// TwinCAT 3 PLC project CNCControl
// ProgramVersion: 3.1.4022.4
// libraries:
//   Tc2_EthernetIP, * (Beckhoff Automation GmbH)
//   Tc2_IoFunctions, * (Beckhoff Automation GmbH)
//   Tc2_Math, * (Beckhoff Automation GmbH)
//   Tc2_Standard, * (Beckhoff Automation GmbH)
//   Tc2_System, * (Beckhoff Automation GmbH)
//   Tc2_Utilities, * (Beckhoff Automation GmbH)
//   Tc3_Module, * (Beckhoff Automation GmbH)
// project tree:
//   DUTs/ E_CIA402State.TcDUT, E_PIDOptimizationStage.TcDUT, E_PIDOptimizationType.TcDUT
//   / EveryHundredMilliseconds.TcTTO, EveryMS.TcTTO (not stored), MainCNCControl.TcTTO (not stored)
//   GVLs/ Constants.TcGVL
//   POUs/ MAIN.TcPOU
//   POUs/SpindleSpeed/ AnalogDemandedSpeedCalculator.TcPOU (not stored), AnalogPrescaledSpeedCalculator.TcPOU, DemandedSpeedInterface.TcIO (not stored), DemandedSpeedTask.TcPOU, PWMDemandedSpeedCalculator.TcPOU, SpindleSpeedCalculator.TcPOU (not stored)
//   POUs/Spindle/ SpindleCIA402Velocity.TcPOU, SpindleController.TcIO, SpindleDeltaVFDOverEIP.TcPOU, SpindleKEBWithEncoder.TcPOU
//   POUs/Utilities/ FB_FreqMeasure.TcPOU, FB_MovingAverageUInt.TcPOU (not stored), FB_MovingAverageReal.TcPOU, FB_OptimizePID.TcPOU (not stored), FB_ScaleBetween.TcPOU (not stored)
//   POUs/Vacuum/ VacuumATV71Ethercat.TcPOU, FB_GetVacuumAMSID.TcPOU, ToshibaP9VacuumPressureGetter.TcPOU, VacuumController.TcIO (not stored)
// real-time tasks:
//   TASK EveryHundredMilliseconds: cycle T#100000us, priority 10, ADS port 350
//   TASK MainCNCControl: cycle T#1ms, priority 6, ADS port 351
//   TASK EveryMS: cycle T#1ms, priority 4, ADS port 352
// I/O:
//   DEVICE Device 1 (EtherCAT), AmsNetId 192.168.1.51.2.1
//     Box 16 (ATV71 EtherCAT) [ATV71 EtherCAT]
//     HITECO UE-1F 6.6 Spindle [KEB_F6_drive_unit_EtherCAT (MDP)]
//       modules: Module 1 (Spindle_Profile)
//     Term 1 (EK1100) [EK1100 EtherCAT Coupler (2A E-Bus)]
//       Term 9 (EL2809) [EL2809 16Ch. Dig. Output 24V, 0.5A]
//       Term 3 (EL1502) [EL1502 2Ch. +/- Counter 24V, 100kHz]
//       Term 4 (EL1809) [EL1809 16Ch. Dig. Input 24V, 3ms]
//       Term 26 (EL6070) [EL6070 1Ch. Licensing-Terminal]
//       Term 17 (EL9110) [EL9110 Power Supplier with LED (24V, Diagnostics)]
//       Term 19 (EL3161) [EL3161 1Ch. Ana. Input 0-10V]
//       Term 12 (EL9011) [EL9011 End Terminal]
//   DEVICE Device 2 (TC3 EIP Scanner), AmsNetId 192.168.1.51.3.1
//     Box 12 (Nitra CMV EtherNet/IP) // <INFO> </INFO> <EDS> C:\TwinCAT\3.1\Config\Io\EtherNetIP\nitraethernetip.eds </EDS>
//     Box 13 (IPE001Z) (disabled) // <INFO> </INFO> <EDS> C:\TwinCAT\3.1\Config\Io\EtherNetIP\IPE001Z_AS1.eds </EDS>
//     Box 2 (CMM-EIP01) (disabled) // <INFO> </INFO> <EDS> C:\TwinCAT\3.1\Config\Io\EtherNetIP\031F000C010400010001.eds </EDS>
// variable links:
//   CNCControl/CNCControl Instance <-> Device 1 (EtherCAT)/Box 16 (ATV71 EtherCAT)
//     MainCNCControl Inputs/MAIN.VacuumControl.iAnalogInput2ScaledValue <-> Inputs/MAIN.VacuumControl.iAnalogInput2ScaledValue
//     MainCNCControl Inputs/MAIN.VacuumControl.iOutputFrequency <-> Inputs/MAIN.VacuumControl.iOutputFrequency
//     MainCNCControl Inputs/MAIN.VacuumControl.iOutputVelocity <-> Inputs/MAIN.VacuumControl.iOutputVelocity
//     MainCNCControl Inputs/MAIN.VacuumControl.iPIDRegulatorFeedback <-> Inputs/MAIN.VacuumControl.iPIDRegulatorFeedback
//     MainCNCControl Inputs/MAIN.VacuumControl.iPIDRegulatorOutput <-> Inputs/MAIN.VacuumControl.iPIDRegulatorOutput
//     MainCNCControl Inputs/MAIN.VacuumControl.iStatusWord <-> Inputs/MAIN.VacuumControl.iStatusWord
//     MainCNCControl Outputs/MAIN.VacuumControl.oMotorFrequency <-> Outputs/MAIN.VacuumControl.oMotorFrequency
//     MainCNCControl Outputs/MAIN.VacuumControl.oVacuumControl <-> Outputs/MAIN.VacuumControl.oVacuumControl
//     MainCNCControl Outputs/MAIN.VacuumControl.oVacuumPressureRequested <-> Outputs/MAIN.VacuumControl.oVacuumPressureRequested
//   CNCControl/CNCControl Instance <-> Device 1 (EtherCAT)/HITECO UE-1F 6.6 Spindle
//     MainCNCControl Inputs/MAIN.SpindleControl.iActualVelocity <-> Module 1 (Spindle_Profile)/Inputs/velocity actual value [0x606C.0]
//     MainCNCControl Inputs/MAIN.SpindleControl.iEncoderErrorState <-> Module 1 (Spindle_Profile)/Inputs/ec01: error encoder interface [0x2801.0]
//     MainCNCControl Inputs/MAIN.SpindleControl.iStatusWord <-> Module 1 (Spindle_Profile)/Inputs/statusword [0x6041.0]
//     MainCNCControl Outputs/MAIN.SpindleControl.oControlWord <-> Module 1 (Spindle_Profile)/Outputs/controlword [0x6040.0]
//     MainCNCControl Outputs/MAIN.SpindleControl.oDigitalInputs <-> Module 1 (Spindle_Profile)/Outputs/di02: dig. input ext. src. [0x3202.0]
//     MainCNCControl Outputs/MAIN.SpindleControl.oTargetVelocity <-> Module 1 (Spindle_Profile)/Outputs/vl target velocity [0x6042.0]
//   CNCControl/CNCControl Instance <-> Device 1 (EtherCAT)/Term 1 (EK1100)/Term 3 (EL1502)
//     EveryHundredMilliseconds Inputs/SpindleSpeedCalculator.CounterValue <-> CNT Inputs Channel 1/Counter value
//   CNCControl/CNCControl Instance <-> Device 1 (EtherCAT)/Term 1 (EK1100)/Term 4 (EL1809)
//     MainCNCControl Inputs/MAIN.iAirPressureSensor <-> Channel 1/MAIN.iPressureSensor
//     MainCNCControl Inputs/MAIN.iS1ToolPresence <-> Channel 5/MAIN.iS1ToolPresence
//     MainCNCControl Inputs/MAIN.iS2ColletOpen <-> Channel 4/MAIN.iS2ColletOpen
//     MainCNCControl Inputs/MAIN.iSpindleOverTemp <-> Channel 3/MAIN.iSpindleOverTemp
//     MainCNCControl Inputs/MAIN.iSpindleToolReleaseButton <-> Channel 2/MAIN.iSpindleToolReleaseButton
//   CNCControl/CNCControl Instance <-> Device 2 (TC3 EIP Scanner)/Box 12 (Nitra CMV EtherNet/IP)
//     MainCNCControl Outputs/MAIN.oValveControl <-> Connection 1 (Input/Output)/Outputs/MAIN.oValveControl

CONFIGURATION CNCControl
    RESOURCE PLC ON TwinCAT3
        TASK EveryHundredMilliseconds(INTERVAL := T#100000us, PRIORITY := 10);
        PROGRAM SpindleSpeedCalculator WITH EveryHundredMilliseconds : SpindleSpeedCalculator;
    END_RESOURCE
END_CONFIGURATION

// ---- DUTs/E_CIA402State.TcDUT
{attribute 'qualified_only'}
{attribute 'strict'}
TYPE E_CIA402State :
(
	Unknown_State,
	NotReadyToSwitchOn,
	SwitchOnDisabled,
	ReadyToSwitchOn,
	SwitchedOn,
	OperationEnabled,
	QuickStopActive,
	FaultReactionActive,
	Fault
);
END_TYPE

// ---- DUTs/E_PIDOptimizationStage.TcDUT
{attribute 'qualified_only'}
{attribute 'strict'}
TYPE E_PIDOptimizationStage :
(
	Init,
	RampingUp,
	RampingDown,
	Done
);
END_TYPE

// ---- DUTs/E_PIDOptimizationType.TcDUT
{attribute 'qualified_only'}
{attribute 'strict'}
TYPE E_PIDOptimizationType :
(
	NoOvershoot,
	SomeOvershoot,
	PessenIntegralRule
);
END_TYPE

// ---- GVLs/Constants.TcGVL
{attribute 'qualified_only'}
VAR_GLOBAL CONSTANT
	// One second in microseconds
	OneSecondInUs : UDINT := 1000000;
END_VAR

// ---- POUs/Spindle/SpindleController.TcIO
INTERFACE SpindleController

// Return the current speed of the spindle in RPM
METHOD GetSpeed : UDINT
VAR_INPUT
END_VAR
END_METHOD

// Start the Spindle running
METHOD Run : BOOL
END_METHOD

// Set the direction the spindle rotates in.
METHOD SetDirection : BOOL
VAR_INPUT
	// Set the spindle rotation direction
	Reverse : BOOL;
END_VAR
END_METHOD

// Set the target speed for the spindle.
METHOD SetSpeed : BOOL
VAR_INPUT
	Speed : UINT;
END_VAR
END_METHOD

// Stop the running spindle
METHOD Stop : BOOL
END_METHOD

END_INTERFACE

// ---- POUs/MAIN.TcPOU
PROGRAM MAIN
VAR
	{region "Air Pressure and Coolant"}
	// Air Pressure >90psi signal to PC pin 10
	oPCAirPressure AT %Q*: BOOL;
	// Air Pressure >90psi signal from sensor.  The sensor triggers as pressure is rising past 90psi
	iAirPressureSensor AT %I*: BOOL;
	// Control of NITRA Valves over ethernet/ip	 
	oValveControl AT %Q* : NitraValves; 
	// Turn on coolant signal from PC
	iPCCoolantOn AT %I* : BOOL;
	{endregion}
	{region "Vacuum"}
	VacuumControl: VacuumATV71Ethercat;
	 // Turn on vacuum signal from PC
	iPCVacuumOn AT %I* : BOOL;
	// Vacuum Pressure good output to PC Pin 7
	oPCVacuumPressureGood AT %Q*: BOOL;
	{endregion}
	{endregion}
	{endregion}
	{region "Spindle variables"}
	{region "Spindle Speed Handling"}
	// True if spindle is at less than 1 RPM
	SpindleStopped : BOOL;
	// Spindle stopped output to PC pin 1
	oPCSpindleStopped AT %Q* : BOOL;
	// Spindle within 5% of speed to PC Pin 28
	oPCSpindleSpeedOK AT %Q* : BOOL;
	{endregion}
	{region "Spindle Tool Change handling"}
	// Tool Release Button on Spindle
	iSpindleToolReleaseButton AT %I*: BOOL;
	// Tool Release from PC Pin 24
	iPCToolRelease AT %I*: BOOL;
	// Tool Presence to PC Pin 2
	oPCToolPresence AT %Q* : BOOL;
	// S1 Tool Presence sensor from the spindle
	iS1ToolPresence AT %I* : BOOL;
	// Collet Open to PC Pin 9
	oPCColletOpen AT %Q* : BOOL;
	// S2 Collet Open sensor from the spindle
	iS2ColletOpen AT %I* : BOOL;	 
	// Spindle over temperature to PC Pin 27
	oPCSpindleOverTemp AT %Q* : BOOL;
	// Spindle over temperature relay
	iSpindleOverTemp AT %I* : BOOL;
	// Turn spindle on input from PC
	iPCSpindleOn AT %I* : BOOL;
	SpindleControl : SpindleKEBWithEncoder;
	{endregion}
	{endregion}
	{region "Input Debouncers"}
	(* The 5V input has a ridiculously fast time - a few nanoseconds.
	   Therefore, we debounce it *)
	CoolantOnDebounced : TON;
	SpindleOnDebounced : TON;
	ToolReleaseDebounced : TON;	
	VacuumOnDebounced : TON;
	{endregion}
END_VAR
VAR CONSTANT
	// Minimum PSI at which vacuum holding is viable for workpiece
	GoodVacuumPressure : REAL := 10.0;
END_VAR

CoolantOnDebounced(IN := iPCCoolantOn, PT := T#3MS);
SpindleOnDebounced(IN := iPCSpindleOn, PT := T#3MS);
ToolReleaseDebounced(IN := iPCToolRelease, PT := T#3MS);
VacuumOnDebounced(IN := iPCVacuumOn, PT := T#3MS);

{region "Probe, Air Pressure, Coolant, Vacuum"}

// Pressure Control
	oPCAirPressure := iAirPressureSensor;

// Coolant control
	oValveControl.Coolant := CoolantOnDebounced.Q;

// Vacuum Control
	IF VacuumOnDebounced.Q THEN
		VacuumControl.Run();
	ELSE 
		VacuumControl.Stop();
	END_IF
	oPCVacuumPressureGood := VacuumControl.GetCurrentPressure() >= GoodVacuumPressure;

{endregion}
{region "Spindle handling"}
// Spindle Speed Handling
	// Spindle is stopped if it is under 1RPM
	SpindleStopped := SpindleSpeedCalculator.SpindleSpeed <= 1.0;
	oPCSpindleStopped := SpindleStopped;
	// Calculate whether spindle is up to speed.  We will only say it is up to speed if it is on.
	oPCSpindleSpeedOK := SpindleOnDebounced.Q AND_THEN (SpindleSpeedCalculator.SpindleSpeed  >= (0.95 * TO_REAL(DemandedSpeedTask.DemandedSpeed)));

// Spindle control handling
	 // NOTE: HSK-F63 spindles may not be spun while the tool is not present
	 IF NOT (SpindleOnDebounced.Q AND iS1ToolPresence) THEN
	 	SpindleControl.SetSpeed(0);
		SpindleControl.Stop();
	 ELSIF SpindleOnDebounced.Q AND iS1ToolPresence THEN	  
	 	SpindleControl.SetSpeed(DemandedSpeedTask.DemandedSpeed);
		SpindleControl.Run();
	 END_IF
		  
// Spindle Tool Change handling
	oPCToolPresence := iS1ToolPresence;
	oPCColletOpen := iS2ColletOpen;
	oPCSpindleOverTemp := iSpindleOverTemp;
	oValveControl.ToolRelease := (iAirPressureSensor AND_THEN SpindleStopped) AND_THEN (ToolReleaseDebounced.Q OR iSpindleToolReleaseButton); 		  

{endregion}		  
{endregion}

END_PROGRAM

// ---- POUs/Vacuum/VacuumATV71Ethercat.TcPOU
FUNCTION_BLOCK VacuumATV71Ethercat IMPLEMENTS  VacuumController
VAR_INPUT
END_VAR
VAR_OUTPUT
END_VAR
VAR
	// Vacuum Control Output
	oVacuumControl AT %Q* : ST_ATV71CommandWord;	
	// Vacuum Pressure requested from VFD - in tenths of a psi from 0 to 1450
	oVacuumPressureRequested AT %Q* : UINT;
		 
	{region "Input Vacuum Data"}
	iStatusWord AT %I* : UINT;
	{attribute 'BaseUnit' := '<RPM, 1, 0, 0>'}
	iOutputVelocity AT %I* : UINT;
	iAnalogInput2ScaledValue AT %I* : UINT;
	{attribute 'UserUnit' := '<Pressure, PSI, PSI, 6894.7572932, 0, centi>'}
	iPIDRegulatorFeedback AT %I* : UINT;
	iPIDRegulatorOutput AT %I* : UINT;
	{attribute 'BaseUnit' := '<Frequency, 0.1, 0, 0>'}
	iOutputFrequency AT %I* : UINT;
	{endregion}
	oMotorFrequency AT %Q* : UINT;
	//	PidOptimizer : FB_OptimizePID;
END_VAR

METHOD GetCurrentPressure : REAL
GetCurrentPressure := TO_REAL(iPIDRegulatorFeedback) / 100;
END_METHOD

METHOD Run : BOOL
oVacuumControl.Forward := TRUE;
oVacuumControl.Reverse := FALSE;
oVacuumControl.PidIntegralOff := FALSE;
	
	(* PID optimization
	IF VacuumOnDebounced.Q THEN
		IF NOT PidOptimizer.TuningDone THEN
			PidOptimizer(Enable := TRUE,
						 ProcessSetpoint := 2500,
						 ProcessValue := iAnalogInput2ScaledValue,
						 NumCycles := 10,
						 Reset := FALSE,
						 ControlLowVal := 5,
						 ControlHighVal := 60,
						 PIDType := E_PIDOptimizationType.FastRamp);
			oMotorFrequency := TO_UINT(PidOptimizer.ControlValue*10);
			IF PidOptimizer.TuningDone THEN
				ADSLOGLREAL(TC2_Utilities.ADSLOG_MSGTYPE_LOG, 'Kp value is %f', PidOptimizer.Kp);
				ADSLOGLREAL(TC2_Utilities.ADSLOG_MSGTYPE_LOG, 'Ki value is %f', PidOptimizer.Ki);
				ADSLOGLREAL(TC2_Utilities.ADSLOG_MSGTYPE_LOG, 'Kd value is %f', PidOptimizer.Kd);
				ADSLOGLREAL(TC2_Utilities.ADSLOG_MSGTYPE_LOG, 'Ku value is %f', PidOptimizer.Ku);
				ADSLOGLREAL(TC2_Utilities.ADSLOG_MSGTYPE_LOG, 'Tu value is %f', PidOptimizer.Tu);
			END_IF
		END_IF
	END_IF
	*)
END_METHOD

METHOD SetPressureRequired : BOOL
VAR_INPUT
	Pressure	: REAL;
END_VAR
oVacuumPressureRequested := TO_UINT(Pressure * 100);
END_METHOD

METHOD Stop : BOOL
oVacuumControl.Forward := FALSE;
oVacuumControl.Reverse := FALSE;
oVacuumControl.PidIntegralOff := FALSE;
END_METHOD

END_FUNCTION_BLOCK

// ---- POUs/Spindle/SpindleKEBWithEncoder.TcPOU
FUNCTION_BLOCK SpindleKEBWithEncoder EXTENDS SpindleCIA402Velocity IMPLEMENTS SpindleController
VAR_INPUT
END_VAR
VAR_OUTPUT
	// This represents the digital inputs of the KEB drive
	// Bit 0 resets the error state
	oDigitalInputs AT %Q* : UINT;
	// Encoder error state
	// Anything other than 0 is an error
	iEncoderErrorState AT %I* : UINT;
END_VAR
VAR
END_VAR

METHOD Stop : BOOL
// The 1024ppr encoder is only good to 12000rpm, so if you go faster, it will get an error that needs to be reset.
// This resets the error state (but only when the spindle is safely stopped)
IF iEncoderErrorState <> 0  AND GetState() = E_CIA402State.SwitchOnDisabled THEN
	oControlWord.FaultReset := TRUE;
ELSE
	oControlWord.FaultReset := FALSE;
	SUPER^.Stop();
END_IF
END_METHOD

END_FUNCTION_BLOCK

// ---- POUs/Spindle/SpindleCIA402Velocity.TcPOU
FUNCTION_BLOCK SpindleCIA402Velocity IMPLEMENTS SpindleController
VAR
	// CIA402 Control word
	oControlWord AT %Q*: ST_CIA402ControlWord;
	// CIA402 Status word
	iStatusWord AT %I*: UINT;
	// CIA402 actual velocity parameter
	iActualVelocity AT %I* : UDINT;
	// CIA402 target velocity
	oTargetVelocity AT %Q* : INT;
	// Forward/backward is specified by positive or negative speed
	VelocityMultiplier : INT := 1;
END_VAR

(* Return the current speed of the spindle in RPM*)
METHOD GetSpeed : UDINT
GetSpeed := iActualVelocity;
END_METHOD

METHOD GetState : E_CIA402State
VAR CONSTANT
	NotReadyToSwitchOnValue : UINT := 2#0000_0000_0000_0000;
	NotReadyToSwitchOnMask : UINT := 2#0000_0000_0100_1111;
	SwitchOnDisabledValue : UINT := 2#0000_0000_0100_0000;
	SwitchOnDisabledMask : UINT := NotReadyToSwitchOnMask;
	ReadyToSwitchOnValue : UINT := 2#0000_0000_0010_0001;
	ReadyToSwitchOnMask : UINT := 2#0000_0000_0110_1111;
	SwitchedOnValue : UINT := 2#0000_0000_0010_0011;
	SwitchedOnMask : UINT := ReadyToSwitchOnMask;
	OperationEnabledValue : UINT := 2#0000_0000_0010_0111;
	OperationEnabledMask : UINT := ReadyToSwitchOnMask;
	QuickStopActiveValue : UINT := 2#0000_0000_0000_0111;
	QuickStopActiveMask : UINT := ReadyToSwitchOnMask;
	FaultReactionActiveValue : UINT := 2#0000_0000_0000_1111;
	FaultReactionActiveMask : UINT := 2#0000_0000_0100_1111;
	FaultValue : UINT := 2#0000_0000_0000_1000;
	FaultMask : UINT := FaultReactionActiveMask;
END_VAR
IF (iStatusWord AND NotReadyToSwitchOnMask) = NotReadyToSwitchOnValue THEN
	GetState := E_CIA402State.NotReadyToSwitchOn;
ELSIF (iStatusWord AND SwitchOnDisabledMask) = SwitchOnDisabledValue THEN
	GetState := E_CIA402State.SwitchOnDisabled;
ELSIF (iStatusWord AND ReadyToSwitchOnMask) = ReadyToSwitchOnValue THEN
	GetState := E_CIA402State.ReadyToSwitchOn;
ELSIF (iStatusWord AND SwitchedOnMask) = SwitchedOnValue THEN
	GetState := E_CIA402State.SwitchedOn;
ELSIF (iStatusWord AND OperationEnabledMask) = OperationEnabledValue THEN
	GetState := E_CIA402State.OperationEnabled;
ELSIF (iStatusWord AND QuickStopActiveMask) = QuickStopActiveValue THEN
	GetState := E_CIA402State.QuickStopActive;
ELSIF (iStatusWord AND FaultReactionActiveMask) = FaultReactionActiveValue THEN
	GetState := E_CIA402State.FaultReactionActive;
ELSIF (iStatusWord AND FaultMask) = FaultValue THEN
	GetState := E_CIA402State.Fault;
ELSE
	GetState := E_CIA402State.Unknown_State;
END_IF
END_METHOD

METHOD GetStatus : ST_CIA402StatusWord
VAR_INPUT
END_VAR
MEMCPY(ADR(GetStatus), ADR(iStatusWord), SIZEOF(iStatusWord));
END_METHOD

METHOD HasFault : BOOL
VAR_INPUT
END_VAR
HasFault := GetState() = E_CIA402State.Fault OR GetState() = E_CIA402State.FaultReactionActive;
END_METHOD

METHOD Run : BOOL
oControlWord.FaultReset := FALSE;
CASE GetState() OF
	E_CIA402State.SwitchOnDisabled:
		oControlWord.EnableVoltage := TRUE;
	E_CIA402State.ReadyToSwitchOn:
		oControlWord.SwitchOn := TRUE;
	E_CIA402State.SwitchedOn:
		oControlWord.EnableOperation := TRUE;
	// We don't need explicit fault handling. 
	// The fault will cause the controller to tell the drive to stop, 
	// and the stop will take care of the fault reset.
END_CASE
END_METHOD

METHOD SetDirection : BOOL
VAR_INPUT
	(* Set the spindle rotation direction*)
	Reverse	: BOOL;
END_VAR
IF Reverse THEN
	VelocityMultiplier := -1;
ELSE
	VelocityMultiplier := 1;
END_IF
END_METHOD

METHOD SetSpeed : BOOL
VAR_INPUT
	Speed	: UINT;
END_VAR
oTargetVelocity := TO_INT(LIMIT(0, Speed, 32767)) * VelocityMultiplier;
END_METHOD

METHOD Stop : BOOL
oControlWord.FaultReset := FALSE;
CASE GetState() OF
	E_CIA402State.SwitchOnDisabled:
		oControlWord.EnableVoltage := FALSE;
		oControlWord.SwitchOn := FALSE;
		oControlWord.EnableOperation := FALSE;
	E_CIA402State.ReadyToSwitchOn:
		oControlWord.EnableVoltage := FALSE;
	E_CIA402State.SwitchedOn:
		oControlWord.SwitchOn := FALSE;
	E_CIA402State.OperationEnabled :
		oControlWord.EnableOperation := FALSE;
	E_CIA402State.Fault : 
		oControlWord.FaultReset := TRUE;
		oControlWord.EnableOperation := FALSE;
		oControlWord.SwitchOn := FALSE;
		oControlWord.EnableVoltage := FALSE;
END_CASE
END_METHOD

END_FUNCTION_BLOCK

// ---- POUs/SpindleSpeed/DemandedSpeedTask.TcPOU
PROGRAM DemandedSpeedTask
VAR
	{attribute 'UserUnit' := '<AngularVelocity, RPM, RPM, 9.549296596425, 0, 0 >'}
	DemandedSpeed : UINT;
	DemandedSpeedImpl : AnalogPrescaledSpeedCalculator;
END_VAR

DemandedSpeed := DemandedSpeedImpl.GetSpeed();

END_PROGRAM

// ---- POUs/SpindleSpeed/AnalogPrescaledSpeedCalculator.TcPOU
// This version uses the EL3161 and it's built in IIR filter
FUNCTION_BLOCK FINAL AnalogPrescaledSpeedCalculator IMPLEMENTS DemandedSpeedInterface; 
VAR_INPUT
	// Analog speed as 0-10v from PC Pin 13
	iAnalogSpeed AT %I*: INT;
END_VAR

METHOD GetSpeed : UINT
GetSpeed := TO_UINT(LIMIT(0, iAnalogSpeed, 24000));
END_METHOD

END_FUNCTION_BLOCK

// ---- POUs/SpindleSpeed/PWMDemandedSpeedCalculator.TcPOU
FUNCTION_BLOCK FINAL PWMDemandedSpeedCalculator IMPLEMENTS DemandedSpeedInterface
VAR
	iInputSpeedBits AT %I* : ARRAY [1..BitArraySize] OF BYTE;
END_VAR
VAR CONSTANT
	// Array Length
	BitArraySize : UINT := 125;
	// PWM frequency
	PWMFrequency : UINT := 200;
    // PWM period
	PWMPeriod : REAL := 1 / PWMFrequency;
	// Microseconds in Frequency
	UsInFrequency : UDINT :=  Constants.OneSecondInUs / PWMFrequency;	
END_VAR

METHOD GetSpeed : UINT
VAR_INST
	TempSpindleSpeed : UINT;
	LastDemandedSpeed : UINT;
	TotalOnTime : UDINT;
	TotalOffTime : UDINT;
	DutyCycle : LREAL;
	DutyCycles : ARRAY [0..20] OF LREAL;
	MovingAverage : FB_MovingAverageReal;
	Scaling : FB_ScaleBetween;
END_VAR
VAR
	I : UINT;	
	J: UINT;
	BitMask : UINT;
	MaskedBit : BOOL;
END_VAR
// The input here is a PWM signal with a frequency of 200, a low of 1% duty, and a high of 95% duty.
// Basic Calculation for PWM pulses

 FOR I := 1 TO BitArraySize BY 1 DO
	 FOR J := 0 TO 7 BY 1 DO
		BitMask := SHL(1, J);
		MaskedBit := TO_BOOL(iInputSpeedBits[I] AND BitMask);
		IF MaskedBit THEN
			TotalOnTime := TotalOnTime + 1;
		ELSE
			TotalOffTime := TotalOffTime + 1; 
		END_IF
		// Stop at the end of the period
		IF (TotalOnTime + TotalOffTime) > UsInFrequency THEN
			EXIT;
		END_IF 
	 END_FOR
 END_FOR
 
// See if the period is up
IF (TotalOnTime + TotalOffTime) > UsInFrequency  THEN
	DutyCycle := TO_LREAL(TotalOnTime) / TO_LREAL(TotalOnTime + TotalOffTime);
	TotalOnTime := 0;
	TotalOffTime := 0;
	// Average the duty cycle and then scale the average
	MovingAverage(ValueToAdd := DutyCycle, 
				  AverageArray := DutyCycles);
	Scaling(RawValue:=MovingAverage.CurrentValue, RawValueMin:=0.0, 
					  RawValueMax:=1, ScaledValueMin:=0,
					  ScaledValueMax:=24000);
	LastDemandedSpeed := TO_UINT(Scaling.ScaledValue);
END_IF
GetSpeed := LastDemandedSpeed;
END_METHOD

END_FUNCTION_BLOCK

// ---- POUs/Utilities/FB_MovingAverageReal.TcPOU
FUNCTION_BLOCK FB_MovingAverageReal
VAR_INPUT
	// Value to add to the moving average.
	ValueToAdd : LREAL;
	// The number of values to store in the array.
	NumValuesToUse : UINT := TO_UINT(UPPER_BOUND(AverageArray, 1) - LOWER_BOUND(AverageArray, 1) + 1);
END_VAR
VAR_IN_OUT
	AverageArray  : ARRAY [*] OF LREAL;
END_VAR
VAR_OUTPUT
	CurrentValue : LREAL;
END_VAR
VAR
	CurrentIndex : UINT;
	NumValuesAdded: UINT;
END_VAR
VAR_TEMP
	Counted : UINT;
	I: DINT;
	Sum: LREAL;
	ArrayLength : UINT := TO_UINT(UPPER_BOUND(AverageArray, 1) - LOWER_BOUND(AverageArray, 1) + 1);
END_VAR

// Compute average over array.
// The order of this addition and MOD are important to avoid going out of bounds.
NumValuesToUse := MIN(ArrayLength, NumValuesToUse);
AverageArray[CurrentIndex] := ValueToAdd;
CurrentIndex := CurrentIndex + 1;
CurrentIndex := CurrentIndex MOD NumValuesToUse;
NumValuesAdded := MIN(NumValuesAdded + 1 , NumValuesToUse);
IF NumValuesAdded > 0 THEN
	FOR I := LOWER_BOUND(AverageArray, 1) TO UPPER_BOUND(AverageArray, 1) BY 1 DO
		Sum := Sum + AverageArray[I];
		Counted := Counted + 1;
		// Don't count more than the number of values.
		IF Counted > NumValuesAdded THEN
			EXIT;
		END_IF
	END_FOR
END_IF
CurrentValue := TO_REAL(Sum / NumValuesAdded);

END_FUNCTION_BLOCK

// ---- POUs/Spindle/SpindleDeltaVFDOverEIP.TcPOU
FUNCTION_BLOCK FINAL SpindleDeltaVFDOverEIP IMPLEMENTS SpindleController
VAR
	// Delta VFD control for the spindle
	oSpindleControl AT %Q* : ST_DeltaVFDCommandWord;
	oSpindleFrequency AT %Q* : UINT;
END_VAR
VAR CONSTANT
	// Number of RPM per HZ in the VFD
	RPMPerHZ : UINT := 30;
	// VFD frequency precision in 1/X of 1 HZ. So 10 means it can do 1/10th of a HZ
	VFDHZPrecision : UINT := 10;
	// Minimum VFD RPM increment based on RPM per HZ and precision
	VFDMinRPMIncrement : UINT := TO_UINT(RPMPerHZ / VFDHZPrecision);
END_VAR

METHOD Run : BOOL
oSpindleControl.Stop := FALSE;
oSpindleControl.Run := TRUE;
END_METHOD

METHOD SetDirection : BOOL
VAR_INPUT
	// Set the spindle rotation direction
	Reverse	: BOOL;
END_VAR
IF Reverse THEN
	oSpindleControl.Reverse := TRUE;
	oSpindleControl.Forward := FALSE;
ELSE
	oSpindleControl.Reverse := FALSE;
	oSpindleControl.Forward := TRUE;
END_IF
END_METHOD

METHOD SetSpeed : BOOL
VAR_INPUT
	Speed: UINT;
END_VAR
// The spindle frequency is in increments of 0.1hz
oSpindleFrequency := (SPEED * Constants.VFDHZPrecision) / Constants.RPMPerHZ;
END_METHOD

METHOD Stop : BOOL
oSpindleControl.Stop := TRUE;
oSpindleControl.Run := FALSE;
END_METHOD

END_FUNCTION_BLOCK

// ---- POUs/Utilities/FB_FreqMeasure.TcPOU
(* This function is the equivalent of FREQ_MEASURE from codesys's utility library.
   It emulates their wacky API that tries to auto-detect specific errors *)
FUNCTION_BLOCK FB_FreqMeasure
VAR_INPUT
	// Input signal
    IN: BOOL;
	// Number of periods to average the frequency over.
	// Must be between 1 and 100
    PERIODS: UINT := 1;
	// Reset all parameters to 0
    RESET: BOOL;
END_VAR
VAR_OUTPUT
	// Frequency in HZ
    OUT: REAL;
	// FALSE until we've measured at least PERIODS periods, or if distance between two rising edges is > 3 * OUT
    VALID: BOOL;
END_VAR
VAR
	RisingEnableEdge: R_TRIG;
	FallingEnableEdge : F_TRIG;
    STARTED: BOOL;
    RISETIME: TIME;
	AveragePeriod : FB_MovingAverageReal;
	// Difference in time between current and last rising edge
    DIFF: DINT;
	// Array of time differences for each period
    TIMEDIFF: ARRAY[0..99] OF LREAL;
	// How many periods we have counted so far
    COUNT: UINT;
	SYSTIMEMS : TIME;          
END_VAR
VAR_TEMP
	OutTemp : LREAL;
END_VAR


IF Reset THEN
    VALID := FALSE;
    COUNT := 0;
    STARTED := FALSE;
    OUT := 0;
    RETURN;
END_IF

RisingEnableEdge(CLK := IN);
FallingEnableEdge(CLK := IN);

(* We care only about whether we are the beginning or the end of the signal.
   If we are at the beginning, we store the current time the signal rose.
   If we are the end, we look at the current time, subtract the rise time,
   and add the signal time period to the period array.
   Once we have collected the requested number of periods, we start averaging
   and mark ourselves valid. *)
IF RisingEnableEdge.Q OR FallingEnableEdge.Q THEN
	// The tming mechanism depends on the PLC. What we expect is something that produces milliseconds.
	// The only requirement is that the difference between the two times represent the signal period in millliseconds
	SYSTIMEMS := ULINT_TO_TIME(F_GetTaskTime() / TC2_Utilities.SYSTEMTIME_TICKSPERMSEC64);
    IF FallingEnableEdge.Q AND STARTED THEN
		DIFF := TIME_TO_DINT(SYSTIMEMS - RISETIME);
		// We assume time never goes backwards for real. Unfortunately, the API of this call does
		// not give us a way to express errors easily.
        IF Diff > 0 THEN
			// Emulate the weird behavior of CODESYS FREQ_MEASURE
			IF VALID AND Diff > 3000 * REAL_TO_DINT(OUT) THEN
				VALID := FALSE;
				COUNT := 0;
				RETURN;
			END_IF
			// Compute moving average over periods
			AveragePeriod(ValueToAdd := DINT_TO_REAL(DIFF),
						  AverageArray := TIMEDIFF,
						  NumValuesToUse := PERIODS,
						  CurrentValue => OutTemp);
			Out := LREAL_TO_REAL (OutTemp); 
            COUNT := MIN(COUNT + 1, PERIODS);
			// Go valid once we have the minimum number of periods to average over.
            VALID := COUNT = PERIODS;
        END_IF
		STARTED := FALSE;
		RETURN;
    END_IF
    STARTED := TRUE;
    RISETIME := SYSTIMEMS;
END_IF

END_FUNCTION_BLOCK

// ---- POUs/Vacuum/FB_GetVacuumAMSID.TcPOU
// This is a very ugly hack because I'm being lazy.
// I'm sure there is some better/more standard way.
FUNCTION_BLOCK FB_GetVacuumAMSID
VAR_INPUT
END_VAR
VAR_OUTPUT
	Busy : BOOL := TRUE;
	VacuumNetID : T_AmsNetID;
END_VAR
VAR
	DoCallOnce : BOOL := TRUE;
	DoOnce : BOOL := TRUE;
	GetLocalAMSId : FB_GetLocalAmsNetId;	

END_VAR
VAR_TEMP
	NetIDLen : INT;
END_VAR

(* We only really want to compute the netid once.
This requires performing the GetLocalAMSId call once and waiting for the result,
and then doing the processing of the result once. *)
IF NOT DoOnce AND NOT DoCallOnce THEN
	RETURN;
END_IF
GetLocalAMSId(bExecute :=  DoCallOnce, tTimeOut := T#5S);
DoCallOnce := FALSE ;
Busy := GetLocalAMSId.bBusy;
IF Busy THEN
	RETURN;
END_IF
IF DoOnce THEN
	DoOnce := FALSE;
	NetIDLen := LEN(GetLocalAMSId.AddrString);
	VacuumNetID := CONCAT(LEFT(GetLocalAMSId.AddrString, NetIDLen-4), '.3.1');
END_IF

END_FUNCTION_BLOCK

// ---- POUs/Vacuum/ToshibaP9VacuumPressureGetter.TcPOU
FUNCTION_BLOCK ToshibaP9VacuumPressureGetter
VAR
	// Vacuum PSI on VFD. The VFD gives it to us without decimal points.
	VacuumPressureFromVFD : WORD;
	// Real Vacuum PSI from 0 to 14.7
	VacuumPressure: REAL;
	GetVacuumPressure : FB_GET_ATTRIBUTE_SINGLE;
	GVPErrorString: STRING(80);
	GetVacuumAMSId : FB_GetVacuumAMSID := ();
END_VAR
VAR CONSTANT
	// This is the application for parameter access on the IPE001Z
	ODVAApplicationObject: WORD := 16#64;
	// FE98 is the VLP pressure monitor register. For monitor variables, we subtract 0x8000 according to the IPE001Z manual
	ToshibaVLPPressureInstance: WORD := TO_WORD(16#FE98) - TO_WORD(16#8000);
END_VAR

// Get the AMS Net ID of the vacuum VFD
GetVacuumAMSId();
IF GetVacuumAMSId.Busy THEN 
	RETURN;
END_IF
// Parameter 
GetVacuumPressure(sNetId := GetVacuumAMSId.VacuumNetID,
		 		  sIPv4Addr := '192.168.1.9',
			  	  bExecute := NOT GetVacuumPressure.bBusy,
				  nClass := ODVAApplicationObject,
				  nInstance := ToshibaVLPPressureInstance,
				  nAttribute := 3,
				  pDst := ADR(VacuumPressureFromVFD),
				  nMaxLen := SIZEOF(VacuumPressureFromVFD));
IF  NOT GetVacuumPressure.bBusy AND GetVacuumPressure.bError THEN
	GVPErrorString := F_GET_ETHERNETIP_ERROR_TEXT(nErrorId := GetVacuumPressure.nErrId);
END_IF
VacuumPressure := TO_REAL(VacuumPressureFromVFD) / 10;

END_FUNCTION_BLOCK
